PROGRAM POU_Master_Calib_1
VAR
	criteria: REAL := 0.5; // Acceptance Criteria (0.1 ~ 5.0)
	failures: INT := 0; // Allowable Failures (0 ~ 5)
	targetVolume: REAL := 0.50; // Volume Target (mL)
	replicates: INT := 5; // Number of checks (0 ~ 10)
	tareWt: REAL; //Weight before
	grossWt: REAL; //Weight after
	netWt: REAL; // rsult of (grossWt - tareWt)
	netVolume: REAL; //result of (netWt * density)
	state: INT;
	valveNo: INT;
	pumpNo: INT:=1;
	timeWt: ton;
	timer2: ton;
	timer3: ton;
	selectPump: ARRAY[1..10] OF STRING;
	result: ARRAY[1..50] OF ST_Results;
	start: BOOL;
	stop: BOOL;
	movimentDONE: BOOL;
	revs: REAL;
	valvePos: USINT;
	repli: INT:= 1;
	axiPower: MC_Power;
	i: INT;
	scale: FB_ScaleDevice;
	adjust: ARRAY[1..10] OF BOOL;
	correctRev: REAL;
	enableAdj: BOOL;
	opening: REAL;
	runLinear: BOOL;
	adjustSum: REAL;
END_VAR

timeWt();
timer2();
timer3();

IF stop THEN
	powerOFF();
	stop:=FALSE;
END_IF

IF pumpNo = 1 OR pumpNo = 2 THEN
	valveNo:= 1;
ELSIF pumpNo = 3 OR pumpNo = 4 THEN
	valveNo:= 2;
ELSIF pumpNo = 5 OR pumpNo = 6 THEN
	valveNo:= 3;
ELSIF pumpNo = 7 OR pumpNo = 8 THEN
	valveNo:= 4;
ELSIF pumpNo = 9 OR pumpNo = 10 THEN
	valveNo:= 5;
END_IF

CASE state OF
	
0: //Idle
	IF start THEN
		GVL_Marco.revs:= GVL_Marco.mL_target;
		GVL_Marco.resetAxi:= FALSE;
		GVL_Marco.valvPos:= 2;
		GVL_Marco.enableValv:= TRUE;
		timeWt(in:=TRUE, pt:=T#10S);
		GVL_Marco.enableAxi:= TRUE;
		FOR i:=1 TO 10 BY 1 DO
			result[i].gross:= 0;
			result[i].rest:= 0;
			result[i].tare:= 0;
		END_FOR
		repli:= 1;
		state:= 10;
	ELSE
		state:= 0;
	END_IF
	
10:	//Enable the pump motor
	
	IF GVL_Motion.aValves[valveNo].Axis.Status.InTargetPosition AND timeWt.Q THEN
		GVL_Marco.enableValv:= FALSE;
		timeWt(in:=FALSE);
		IF pumpNo >= 10 THEN
			pumpNo:= 2;
			state:= 20;
		ELSE
			pumpNo:= pumpNo + 1;
			state:= 0;
		END_IF
	ELSE
		state:= 10;
	END_IF		

20:	//Fill the Jars from Bottle
	
	IF NOT GVL_Motion.aPumps[pumpNo].Rotary.Axis.Status.Disabled AND timer2.Q THEN
		revs:= GVL_Marco.revs*2.4;
		GVL_Marco.runFWD:= TRUE;
		timer2(in:=TRUE, pt:=T#10S);
		IF pumpNo >= 10 THEN
			pumpNo:= 2;
			start:= FALSE;
			state:= 30;
		ELSE
			timer2(in:=FALSE);
			pumpNo:= pumpNo + 1;
			GVL_Marco.runFWD:= FALSE;
			state:= 20;
		END_IF
	ELSE
		state:= 20;
	END_IF

30: //Move valve to position 6
	
	IF NOT GVL_Motion.aPumps[pumpNo].Rotary.Axis.Status.Moving AND timer2.Q THEN
		GVL_Marco.runFWD:= FALSE;
		GVL_Marco.valvPos:= 6;
		GVL_Marco.enableValv:= TRUE;
		timer2(in:=FALSE);
		timeWt(in:=TRUE, pt:=T#10S);
		IF pumpNo >= 10 THEN
			pumpNo:= 2;
			state:= 40;
		ELSE
			pumpNo:= pumpNo + 1;
			state:= 30;
		END_IF
	ELSE
		state:= 30;
	END_IF


40: //Fill the calibration box( SETUP )

	IF GVL_Motion.aValves[valveNo].Axis.Status.InTargetPosition AND timeWt.Q THEN
		GVL_Marco.enableValv:= FALSE;
		revs:= GVL_Marco.revs/2;
		GVL_Marco.runBWD:= TRUE;
		timeWt(in:=FALSE);
		timer2(in:=TRUE, pt:=T#5S);
		state:= 50;
		
	ELSE
		state:= 40;	
	END_IF

50: //Waiting

	IF NOT GVL_Motion.aPumps[pumpNo].Rotary.Axis.Status.Moving AND timer2.Q THEN
		GVL_Marco.runBWD:= FALSE;
		timer2(in:=FALSE);
		timeWt(in:=TRUE, pt:=T#10S);
		GVL_Calibration.fbScaleDevice.RequestWeight();
		state:= 55;
	ELSE
		state:= 50;
	END_IF
	
55: //Make Tara
	
	IF timeWt.Q THEN
		tareWt:= GVL_Calibration.fbScaleDevice.RequestWeight();
		timeWt(in:=FALSE);
		state:= 60;
	ELSE
		state:= 55;
	END_IF
	
60: //Fill calibration box

	IF tareWt <> 9999.0 THEN
		result[repli].tare:= tareWt;
		revs:= GVL_Marco.revs;
		GVL_Marco.runBWD:= TRUE;
		timer2(in:=TRUE, pt:=T#5S);
		state:= 70;
	ELSE
		state:= 60;
	END_IF
	
70: //Waiting

	IF NOT GVL_Motion.aPumps[pumpNo].Rotary.Axis.Status.Moving AND timer2.Q THEN
		GVL_Marco.runBWD:= FALSE;
		timer2(in:=FALSE);
		timeWt(in:=TRUE, pt:=T#10S);
		GVL_Calibration.fbScaleDevice.RequestWeight();
		state:= 75;
	ELSE
		state:= 70;
	END_IF

75: //Get gross weight
	
	IF timeWt.Q THEN
		grossWt:= GVL_Calibration.fbScaleDevice.RequestWeight();
		timeWt(in:=FALSE);
		state:= 80;
	ELSE
		state:= 75;
	END_IF
	
80: //Return solvent to jar

	IF grossWt <> 9999.0 THEN
		result[repli].gross:= grossWt;
		result[repli].rest:= result[repli].gross - result[repli].tare;
		netWt:= result[repli].rest;
			IF (netWt > GVL_Marco.mL_target+((GVL_Marco.mL_target*0.5)/100) OR netWt < GVL_Marco.mL_target-((GVL_Marco.mL_target*0.5)/100)) THEN
				adjust[repli]:= TRUE;
			ELSE
				adjust[repli]:= FALSE;
			END_IF
			IF repli >= replicates THEN
				revs:= GVL_Marco.revs*2;
				GVL_Marco.runFWD:= TRUE;
			ELSE
				revs:= GVL_Marco.revs;
				GVL_Marco.runFWD:= TRUE;
			END_IF
		timer3(in:=TRUE, pt:=T#10S);
		repli := repli +1;
		state:= 90;
	ELSE
		state:= 80;
	END_IF

90: //Check replicates

	IF repli < replicates+1 AND timer3.Q AND GVL_Motion.aPumps[pumpNo].Rotary.Axis.Status.NotMoving THEN
		timer3(in:=FALSE);
		GVL_Marco.runFWD:= FALSE;
		timer2(in:=TRUE, pt:=T#5S);
		state:= 50;
	ELSIF repli >= replicates AND timer3.Q AND GVL_Motion.aPumps[pumpNo].Rotary.Axis.Status.NotMoving THEN
		timer3(in:=FALSE);
		GVL_Marco.runFWD:= FALSE;
		GVL_Marco.valvPos:= 2;
		GVL_Marco.enableValv:= TRUE;
		timer2(in:=TRUE, pt:=T#10S);
		IF pumpNo >= 10 THEN
			pumpNo:= 2;
			state:= 100;
		ELSE
			pumpNo:= pumpNo + 1;
			repli:= 1;
			state:= 50;
		END_IF
	ELSE
		state:= 90;
	END_IF

100: //Empty the jar

	IF  GVL_Motion.aValves[valveNo].Axis.Status.InTargetPosition AND timer2.Q THEN
		GVL_Marco.enableValv:= FALSE;
		revs:= GVL_Marco.revs*2.4;
		GVL_Marco.runBWD:= TRUE;
		timer2(in:=FALSE);
		timer3(in:=TRUE, pt:=T#10S);
		IF pumpNo >= 10 THEN
			pumpNo:= 2;
			state:= 110;
		ELSE
			pumpNo:= pumpNo + 1;
			state:= 100;
		END_IF
	ELSE
		state:= 100;
	END_IF
	
110: //Done

	IF NOT GVL_Motion.aPumps[pumpNo].Rotary.Axis.Status.Moving AND timer3.Q THEN
		GVL_Marco.runBWD:= FALSE;
		timer3(in:=FALSE);
		timeWt(in:=TRUE, pt:=T#10S);
		IF pumpNo >= 10 THEN
			pumpNo:= 2;
			state:= 120;
		ELSE
			pumpNo:= pumpNo + 1;
			state:= 110;
		END_IF
	ELSE
		state:= 110;
	END_IF
	
120:

	IF GVL_Motion.aPumps[pumpNo].Rotary.Axis.Status.NotMoving AND timeWt.Q THEN
		GVL_Marco.resetAxi:= TRUE;
		GVL_Marco.enableAxi:= FALSE;
		IF pumpNo >= 10 THEN
			pumpNo:= 2;
			state:= 0;
		ELSE
			pumpNo:= pumpNo + 1;
			state:= 120;
		END_IF
	ELSE
		state:= 120;
	END_IF
	
END_CASE

METHOD moveValve : BOOL
VAR
	state: INT;
	valveNo: INT;
END_VAR
VAR_INPUT
	pumNo: INT;
	valvePos: USINT;
	
END_VAR
IF pumpNo = 1 OR pumpNo = 2 THEN
	valveNo:= 1;
ELSIF pumpNo = 3 OR pumpNo = 4 THEN
	valveNo:= 2;
ELSIF pumpNo = 5 OR pumpNo = 6 THEN
	valveNo:= 3;
ELSIF pumpNo = 7 OR pumpNo = 8 THEN
	valveNo:= 4;
ELSIF pumpNo = 9 OR pumpNo = 10 THEN
	valveNo:= 5;
END_IF

GVL_Motion.aValvesObj[valveNo].MoveValve(iPosition := valvePos, rVelocity := GVL_Motion.aValves[1].rTargetVel, rAcc := GVL_Motion.aValves[1].rAcceleration, rDec := GVL_Motion.aValves[1].rDeceleration);

CASE state OF
	
0:

	IF NOT GVL_Motion.aValves[valveNo].Axis.Status.Moving THEN
		GVL_Motion.aValvesObj[valveNo].MoveValve(iPosition := valvePos, rVelocity := GVL_Motion.aValves[1].rTargetVel, rAcc := GVL_Motion.aValves[1].rAcceleration, rDec := GVL_Motion.aValves[1].rDeceleration);
		movimentDONE:=FALSE;
		state:= 1;
	ELSE
		state:= 0;	
	END_IF

1:
	IF NOT GVL_Motion.aValves[valveNo].Axis.Status.Moving THEN
			movimentDONE:= TRUE;
			State:= 0;
		ELSE
			state:= 1;
		END_IF
	
	
END_CASE
END_METHOD

METHOD powerOFF : BOOL
VAR
	axiPower: MC_Power;
	pumpNo: INT;
	
END_VAR
VAR_INPUT
	
	
END_VAR
FOR pumpNo:=1 TO 10 BY 1 DO
	axiPower(
	Axis:= GVL_Motion.aPumps[pumpNo].Rotary.Axis,
	Enable:= FALSE,
	Enable_Negative:= FALSE,
	Enable_Positive:= FALSE,
	Override:= 100);
	
	axiPower(
	Axis:= GVL_Motion.aPumps[pumpNo].Linear.Axis,
	Enable:= FALSE,
	Enable_Negative:= FALSE,
	Enable_Positive:= FALSE,
	Override:= 100);
END_FOR
END_METHOD

METHOD runBwd : BOOL
VAR
	moveRel: MC_MoveRelative;
	selectPosRel: LREAL;
	
END_VAR
VAR_INPUT
	pumpNo: INT;
	revs: INT;
	 
END_VAR

selectPosRel:= revs*360;

moveRel(
	Axis:= GVL_Motion.aPumps[pumpNo].Rotary.Axis,
	Execute:= TRUE,
	Distance:= selectPosRel*-1,
	Velocity:= 3000,
	Acceleration:= 3000,
	Deceleration:= 3000);
END_METHOD

METHOD runFwd : BOOL
VAR
	moveRel: MC_MoveRelative;
	selectPosRel: LREAL;
	
END_VAR
VAR_INPUT
	pumpNo: INT;
	revs: INT;
	 
END_VAR

selectPosRel:= revs*360;

moveRel(
	Axis:= GVL_Motion.aPumps[pumpNo].Rotary.Axis,
	Execute:= TRUE,
	Distance:= selectPosRel,
	Velocity:= 3000,
	Acceleration:= 3000,
	Deceleration:= 3000);
END_METHOD

END_PROGRAM

(* stored: Version 1.1.0.1, ProductVersion 3.1.4024.15
   POU POU_Master_Calib_1: Id {20f3d9b9-1bf2-45a4-9598-b97882a704d8}, SpecialFunc None
   Method moveValve: Id {eeb6051d-fdc9-4533-bd58-1682f85fdb08}
   Method powerOFF: Id {252a9145-3840-459e-b3fa-36a7b798bd8e}
   Method runBwd: Id {e08c0703-be6f-4c54-b395-f033178d74ad}
   Method runFwd: Id {57ca53e5-03a8-4969-b9c4-a9a5d21b1dbd} *)
